// TIA Portal V19 export
TYPE "type_xyzResponsetData"
// stored: Access Published, Namespace Unit3
   STRUCT
      u1XyzEnabled : Bool;   // 是否允许运动
      u2XyzEnabled : Bool;   // 是否允许运动
   END_STRUCT;
END_TYPE
